{attribute 'qualified_only'}
{attribute 'to_string'}
TYPE E_GCServiceId :
(
	// Each value identifies one Service instance within the GC Module.
	None := 0,
	SpinAxisJogCW := 1,
	SpinAxisMoveAbs := 2,
	SpinAxisMoveVelCW := 3,
	LiftPinAxisMoveVelCW := 4,
	LiftPinAxisMoveVelCCW := 5,
	LiftPinAxisMoveAbs := 6,
	SingleProcess := 7,
	WaferSend := 8,
	WaferReceive := 9
) UDINT;
END_TYPE

(* stored: Version 1.1.0.1, ProductVersion 3.1.4026.18
   DUT E_GCServiceId: Id {c093ca56-3521-4ff1-9f31-1d625a170479} *)
